// TIA Portal V18 export
TYPE "RCS_KeyenceSR1000_HMI1"
// stored: IsFailsafeCompliant false
   STRUCT
      Manual : Struct
         Preset : Bool;
         Trigger : Bool;
      END_STRUCT;
      Status : Struct
         Ready : Bool;
         Busy : Bool;
         Failure : Bool;
         Complete : Bool;
         ReadOk : Bool;
         ReadNok : Bool;
         TimeOut : Bool;
         Error : Bool;
         ErrorCode : UInt;
         Sequence : Int;
         iReTriggerTimes : USInt;
         CurrentLength : UInt;
         CurrentCode : String[128];
         LastCode : String[128];
      END_STRUCT;
      Indata : Struct
         ReadComplete : Bool;
         ReadFailure : Bool;
         GeneralErrorCode : UInt;
         ReadResultCode : UInt;
         ResultDataSize : UInt;
      END_STRUCT;
      Outdata : Struct
         ReadCompleteClear : Bool;
         ErrorClear : Bool;
         ReadRequest : Bool;
      END_STRUCT;
   END_STRUCT;
END_TYPE
